FUNCTION_BLOCK OnePumpFF_Latch
VAR_INPUT
	DP_Switch: BOOL;
	Pump_Run: BOOL;
	OA_AlarmReset: BOOL;
	PumpFailureDelay: TIME;
END_VAR
VAR_OUTPUT
	PumpFlow_Alarm: BOOL;
END_VAR
VAR
	NoFlow: BOOL;
	T1: TON;
END_VAR

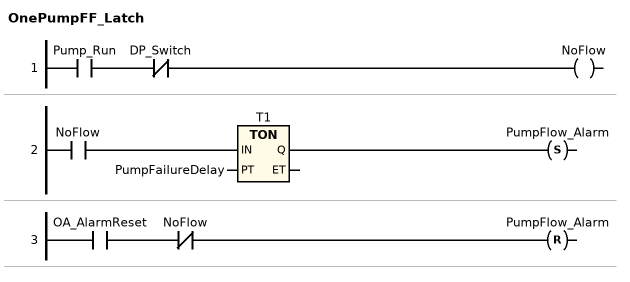
// NETWORK 1
NoFlow := Pump_Run AND NOT DP_Switch;

// NETWORK 2
T1(IN := NoFlow, PT := PumpFailureDelay); // TON
PumpFlow_Alarm S= T1.Q;

// NETWORK 3
PumpFlow_Alarm R= OA_AlarmReset AND NOT NoFlow;

END_FUNCTION_BLOCK

(* stored: Version 1.1.0.1, ProductVersion 3.1.4024.12
   POU OnePumpFF_Latch: Id {74c2989e-70f0-470e-92b5-1b94ddd38823}, SpecialFunc None *)
